Yaskawa INFORM job: OK_R2_O55A(90,180)KMOK_HARDOX.JBI

/JOB
//NAME OK_R2_O55A(90,180)KMOK_HARDOX
//POS
///NPOS 281,281,281,21,0,0
///TOOL 0
///POSTYPE PULSE
///PULSE
C00000=-111506,-49155,-65609,8484,85356,-77443
C00001=-115517,55698,23689,9444,84726,-78820
C00002=-108924,22008,-28178,-1197,90006,-78517
C00003=-108800,12121,-29647,4496,81806,-65930
C00004=-108630,12702,-28416,4432,81339,-65891
C00005=-108630,12328,-27828,4436,80786,-65911
C00006=-108630,12408,-27956,4436,80905,-65905
C00007=-108261,14534,-26027,4289,80792,-65794
C00008=-108630,12408,-27956,4436,80905,-65905
C00009=-107811,11629,-28656,4106,80897,-65648
C00010=-106858,10805,-29394,3723,80886,-65349
C00011=-107811,12739,-30286,4093,82467,-65597
C00012=-109010,42723,-6645,1454,97503,-73185
C00013=-109059,41996,-5623,1462,96501,-73210
C00014=-109059,41520,-5019,1461,95884,-73214
C00015=-109059,41606,-5129,1461,95997,-73214
C00016=-109349,39393,-7454,1528,96295,-73302
C00017=-109059,41606,-5129,1461,95997,-73214
C00018=-105960,29621,-15205,-5152,89122,-73169
C00019=-106826,30438,-14390,-4880,88993,-73434
C00020=-106699,31092,-15669,-4922,90120,-73439
C00021=-111304,-6970,-55605,-8918,107850,-76513
C00022=-101629,-20179,-65627,-10374,108234,-73505
C00023=-102461,-22935,-63329,-10075,105355,-73520
C00024=-102461,-23546,-62650,-10036,104633,-73460
C00025=-102461,-23453,-62757,-10042,104746,-73469
C00026=-102879,-26170,-64656,-9970,104475,-73577
C00027=-102461,-23453,-62757,-10042,104746,-73469
C00028=-99476,-55184,-78355,-14129,83990,-71244
C00029=-100829,-54344,-77892,-13696,83914,-71680
C00030=-99476,-54678,-79370,-14114,84849,-71342
C00031=-104557,-74568,-89383,-2164,74355,-70375
C00032=-103806,-74176,-87211,-2482,73240,-70100
C00033=-103806,-74372,-86383,-2489,72630,-70088
C00034=-103806,-74333,-86558,-2489,72756,-70088
C00035=-103548,-71014,-84973,-2584,73493,-70016
C00036=-103806,-74333,-86558,-2489,72756,-70088
C00037=-102597,-74952,-86848,-2986,72658,-69674
C00038=-101312,-75790,-87238,-3514,72521,-69232
C00039=-102597,-74499,-88609,-2967,73972,-69706
C00040=-118555,-42842,-73429,3462,80943,-74869
C00041=-119429,-43574,-71478,3824,79408,-75190
C00042=-119429,-43990,-70690,3831,78712,-75212
C00043=-119429,-43899,-70866,3830,78866,-75207
C00044=-122277,-43888,-70860,4961,79012,-76114
C00045=-122277,-44025,-70591,4964,78778,-76124
C00046=-121086,-44057,-70608,4493,78709,-75744
C00047=-121531,-43284,-72024,4653,79998,-75839
C00048=-117272,-117266,-105575,3266,62469,-74939
C00049=-116519,-127007,-107880,3037,58859,-74752
C00050=-116519,-126380,-106487,3053,58326,-74766
C00051=-116519,-126568,-106901,3048,58484,-74761
C00052=-121865,-126759,-106958,5473,58705,-76855
C00053=-121865,-126441,-106262,5489,58442,-76869
C00054=-119655,-126444,-106264,4491,58305,-76004
C00055=-119655,-127215,-107960,4461,58951,-75978
C00056=-112812,-150066,-114118,1491,50753,-73411
C00057=-112812,-148729,-112487,1496,50436,-73414
C00058=-113217,-142059,-110816,1647,52843,-73550
C00059=-113131,-144600,-112664,1608,52672,-73518
C00060=-64818,-116281,-103066,-23997,61655,-54736
C00061=-62465,-114100,-100180,-25084,61755,-53781
C00062=-62465,-113608,-98707,-25230,61158,-53639
C00063=-62465,-113710,-99005,-25201,61277,-53666
C00064=-58836,-120022,-101046,-27063,60627,-51963
C00065=-58836,-119826,-100588,-27108,60466,-51920
C00066=-60233,-117500,-99850,-26399,60681,-52575
C00067=-60033,-118628,-101973,-26303,61399,-52670
C00068=-95049,-20989,-71107,5943,107094,-67526
C00069=-77423,-912,-56771,2322,107833,-62256
C00070=-76072,-2112,-53613,2004,105243,-61899
C00071=-76072,-2916,-53031,1997,104470,-61910
C00072=-76072,-2789,-53124,1997,104594,-61910
C00073=-75971,-5189,-55074,1975,104559,-61882
C00074=-76072,-2789,-53124,1997,104594,-61910
C00075=-72991,-17697,-62638,-2229,94769,-69319
C00076=-74281,-17927,-62808,-1837,94727,-69700
C00077=-72991,-16562,-63565,-2235,95923,-69339
C00078=-75226,-46418,-75690,9290,73375,-84742
C00079=-74182,-46690,-75145,8802,72795,-84444
C00080=-74182,-47182,-74296,8836,72029,-84500
C00081=-74182,-47096,-74453,8830,72169,-84490
C00082=-74244,-44038,-72629,8839,72620,-84478
C00083=-74182,-47096,-74453,8830,72169,-84490
C00084=-73094,-46764,-74257,8291,72112,-84135
C00085=-72074,-46719,-74230,7784,72025,-83806
C00086=-72401,-46093,-76320,7882,73648,-83808
C00087=-67489,-6166,-61905,14115,111060,-76264
C00088=-69649,20522,-33673,24556,114676,-73904
C00089=-69671,18738,-32349,24199,113097,-74275
C00090=-69671,18146,-31824,24077,112524,-74402
C00091=-69671,18262,-31932,24102,112638,-74377
C00092=-69800,17846,-32320,24118,112695,-74410
C00093=-69675,18599,-32561,24211,113152,-74264
C00094=-63225,2541,-47955,23753,112661,-72111
C00095=-63277,1683,-47440,23617,111977,-72278
C00096=-63277,1073,-46916,23502,111394,-72405
C00097=-63277,1203,-47030,23526,111518,-72377
C00098=-63425,725,-47430,23545,111556,-72420
C00099=-63342,1826,-48065,23712,112415,-72205
C00100=-62206,17260,-37784,17009,103305,-74838
C00101=-61339,16149,-35110,16634,101032,-74890
C00102=-61339,15490,-34544,16589,100372,-74981
C00103=-61339,15587,-34628,16595,100471,-74968
C00104=-60359,16269,-33999,16356,100262,-74691
C00105=-61339,15587,-34628,16595,100471,-74968
C00106=-61066,13263,-36755,16538,100533,-74873
C00107=-60785,11321,-38512,16476,100561,-74782
C00108=-61066,13913,-37304,16583,101180,-74784
C00109=-55537,11439,-40793,10264,96708,-89931
C00110=-55386,12069,-40617,10225,96903,-89870
C00111=-55386,11332,-40052,10205,96188,-89929
C00112=-55386,11448,-40144,10209,96302,-89918
C00113=-56455,10727,-40790,10532,96446,-90224
C00114=-55386,11448,-40144,10209,96302,-89918
C00115=-55615,12989,-38751,10276,96262,-89989
C00116=-56013,15101,-36821,10392,96204,-90111
C00117=-55930,15302,-38056,10390,97045,-90015
C00118=-69610,-27139,-66329,21663,80743,-86076
C00119=-68739,-29162,-64945,21405,78779,-86142
C00120=-68739,-29645,-64290,21446,78173,-86252
C00121=-68739,-29425,-64595,21426,78455,-86201
C00122=-70305,-29836,-64873,22111,78793,-86664
C00123=-70305,-30098,-64507,22135,78458,-86726
C00124=-69784,-29812,-64314,21908,78356,-86568
C00125=-70093,-29888,-65249,22006,78930,-86565
C00126=-69460,-16189,-57169,21614,80708,-86031
C00127=-69490,-16804,-56284,21674,79908,-86184
C00128=-69490,-17306,-55650,21712,79303,-86294
C00129=-69490,-16804,-56284,21674,79908,-86184
C00130=-71198,-17146,-56538,22415,80299,-86675
C00131=-71198,-17694,-55840,22455,79641,-86800
C00132=-70522,-17552,-55735,22163,79484,-86605
C00133=-70652,-17250,-56551,22180,80125,-86528
C00134=-59067,-8187,-54664,-1101,82113,-86494
C00135=-58982,-12091,-55682,-1142,80734,-86460
C00136=-58982,-12659,-55089,-1143,80077,-86456
C00137=-58982,-12365,-55400,-1142,80420,-86459
C00138=-58542,-15777,-57986,-1343,80263,-86324
C00139=-58542,-16216,-57517,-1344,79752,-86321
C00140=-58731,-14747,-56416,-1258,79827,-86379
C00141=-58929,-14817,-58024,-1165,80777,-86449
C00142=-74865,-14118,-62828,-14130,92718,-81050
C00143=-74988,-16459,-62145,-14059,91123,-80906
C00144=-74988,-17205,-61497,-14051,90361,-80819
C00145=-74988,-16814,-61843,-14056,90763,-80864
C00146=-74878,-20571,-64590,-14091,90545,-80806
C00147=-74878,-21004,-64202,-14087,90099,-80754
C00148=-75042,-19403,-63044,-14030,90184,-80814
C00149=-74977,-18175,-64416,-14070,91627,-80958
C00150=-70693,-7790,-53035,631,77874,-74575
C00151=-70154,-9444,-51202,364,75895,-74417
C00152=-70154,-9889,-50670,365,75339,-74418
C00153=-70154,-9794,-50790,365,75461,-74418
C00154=-70309,-7210,-48753,442,75536,-74465
C00155=-70154,-9794,-50790,365,75461,-74418
C00156=-69601,-9613,-50649,89,75466,-74246
C00157=-68418,-9035,-50194,-503,75489,-73877
C00158=-70154,-8777,-51949,363,76695,-74414
C00159=-72134,44695,-6984,-4762,104287,-75834
C00160=-72134,44301,-6603,-4750,103850,-75816
C00161=-72134,43688,-5973,-4734,103152,-75788
C00162=-72134,43787,-6082,-4735,103269,-75794
C00163=-72123,41447,-8571,-4742,103595,-75805
C00164=-72134,43787,-6082,-4735,103270,-75794
C00165=-73005,43598,-6282,-4599,103251,-76067
C00166=-73786,43384,-6510,-4475,103242,-76313
C00167=-73018,44528,-7213,-4622,104298,-76111
C00168=-79422,35817,-13411,7006,100751,-75778
C00169=-74570,36341,-12845,6044,100322,-74293
C00170=-74570,36341,-12845,6044,100322,-74293
C00171=-72929,24013,-22984,4225,91927,-74293
C00172=-70584,14325,-29595,-1089,84518,-74676
C00173=-68494,21486,-24488,-6892,89276,-75326
C00174=-69395,21903,-23934,-10573,89960,-76456
C00175=-69395,21903,-23934,-10573,89960,-76456
C00176=-71080,32446,-16078,-8958,97674,-77386
C00177=-79422,35817,-13411,7006,100751,-75778
C00178=-79438,36883,-13685,7031,101465,-75742
C00179=-62206,17260,-37784,17009,103305,-74838
C00180=-61339,16149,-35110,16634,101032,-74890
C00181=-60712,-19322,-56729,15368,77567,-77605
C00182=-59094,-21751,-57339,14674,76450,-77219
C00183=-61038,-23011,-55706,17436,71746,-78177
C00184=-62083,-14156,-49199,17905,72476,-78422
C00185=-62083,-14156,-49199,17905,72476,-78422
C00186=-57090,11564,-36742,7182,90651,-76876
C00187=-56002,36932,-16764,6614,106870,-88572
C00188=-52140,41844,-13688,6040,107237,-87347
C00189=-48975,42648,-12828,5535,106926,-86378
C00190=-48975,42648,-12828,5535,106926,-86378
C00191=-52691,32805,-21114,13853,102301,-85620
C00192=-59094,-21751,-57339,14674,76450,-77219
C00193=-59425,-21539,-59164,14761,77698,-77175
C00194=-82076,-56968,-83798,24635,79831,-84346
C00195=-77747,-24152,-67705,18938,100689,-79924
C00196=-78057,-28160,-69137,18928,99634,-80190
C00197=-70869,-26802,-68287,17174,98411,-78082
C00198=-70869,-26802,-68287,17174,98411,-78082
C00199=-62364,-43762,-77635,6437,85665,-78480
C00200=-58442,-42143,-76885,-289,85725,-78490
C00201=-56915,-39089,-75695,-4701,88717,-80179
C00202=-58604,-34961,-73950,-7014,92707,-81523
C00203=-58604,-34961,-73950,-7014,92707,-81523
C00204=-58166,-35258,-74455,-8537,94295,-81804
C00205=-78057,-28160,-69137,18928,99634,-80190
C00206=-78109,-26468,-70352,19060,101178,-79960
C00207=-101629,-20179,-65627,-10374,108234,-73505
C00208=-103344,-22647,-63272,-9953,105369,-73804
C00209=-103510,-25764,-64254,-9875,104364,-73776
C00210=-96684,-29558,-66841,-10807,104795,-71624
C00211=-96684,-29558,-66841,-10807,104795,-71624
C00212=-95283,-51624,-78295,-10520,89912,-69715
C00213=-89288,-71016,-83236,-19331,74161,-66844
C00214=-92735,-73848,-83866,-17944,70715,-67525
C00215=-98754,-71520,-82752,-15362,70010,-69594
C00216=-98754,-71520,-82752,-15362,70010,-69594
C00217=-103983,-45462,-74593,-9714,90020,-72843
C00218=-103510,-25764,-64254,-9875,104364,-73776
C00219=-103560,-24307,-64999,-9933,105549,-73890
C00220=-69649,20522,-33673,24556,114676,-73904
C00221=-71557,26749,-25386,24354,113424,-74867
C00222=-68289,18895,-32791,17896,110504,-75619
C00223=-68202,19061,-32635,17883,110476,-75594
C00224=-68581,18341,-33310,17936,110593,-75702
C00225=-67453,16954,-34605,17788,110459,-75347
C00226=-67453,17755,-35235,17895,111222,-75226
C00227=-59289,756,-51060,6867,103388,-84120
C00228=-56748,-5812,-54346,2389,98605,-84475
C00229=-64645,12200,-39595,15963,109468,-83302
C00230=-61225,2939,-46046,22972,113017,-79913
C00231=-60681,1709,-47088,22917,112895,-79749
C00232=-58469,-3087,-51074,22687,112356,-79091
C00233=-58469,-1901,-52028,22910,113464,-78859
C00234=-117837,-87974,-96376,3289,71861,-74881
C00235=-92533,-132854,-111618,-21009,63789,-66049
C00236=-78523,-139004,-102182,-39306,54450,-56561
C00237=-81657,-141710,-102852,-38814,52284,-57229
C00238=-81657,-141710,-102852,-38814,52284,-57229
C00239=-114174,-154940,-107271,-2509,34053,-71746
C00240=-140780,-145696,-102896,33687,43289,-86686
C00241=-138023,-130656,-99106,29500,46903,-83798
C00242=-128713,-21741,-47637,18171,66698,-75148
C00243=-128713,-20196,-51555,17794,69753,-74669
C00244=-109059,43195,-6970,1468,97945,-73193
C00245=-113001,46227,-1101,7447,98334,-73296
C00246=-113396,48521,2242,7746,99771,-73296
C00247=-109170,43506,-3227,7034,100204,-71930
C00248=-109170,43506,-3227,7034,100204,-71930
C00249=-110675,25111,-18338,12830,89041,-80433
C00250=-106850,7079,-30449,5687,75314,-81784
C00251=-105360,10734,-28025,177,76815,-82287
C00252=-108676,13612,-25432,1655,76734,-83345
C00253=-108676,13612,-25432,1655,76734,-83345
C00254=-107152,30192,-14315,-2638,88634,-83622
C00255=-113396,48521,2242,7746,99771,-73296
C00256=-113396,49658,801,7791,101229,-73204
C00257=-101766,-98767,-99644,-3411,68336,-69273
C00258=-70067,-34207,-71053,21900,80175,-86329
C00259=-68941,-37910,-69134,21595,77036,-86529
C00260=-69099,-37316,-68757,21658,77143,-86564
C00261=-69654,-30548,-64331,21843,77979,-86598
C00262=-70579,-15119,-53564,22144,79419,-86640
C00263=-70579,-15119,-53564,22144,79419,-86640
C00264=-59362,-1592,-48978,2748,88384,-85470
C00265=-54202,-4221,-50196,-5979,86559,-88824
C00266=-54998,-5045,-50841,-6864,86759,-89370
C00267=-54493,-339,-47792,-12989,90949,-86203
C00268=-70768,-8822,-54873,-7152,89179,-90922
C00269=-60817,-19294,-55988,-26592,80523,-79978
C00270=-60817,-16249,-59555,-26407,83905,-80744
C00271=-62218,-50547,-80619,-18317,72013,-76735
C00272=-117272,-117266,-105575,3266,62469,-74939
C00273=-127230,-85492,-91646,16880,70768,-77338
C00274=-127349,-94743,-89409,19343,58411,-79334
C00275=-124353,-95100,-89551,17820,57640,-78233
C00276=-84234,-78954,-82744,-5379,58597,-62424
C00277=-80328,-74945,-80894,-7540,59821,-60991
C00278=-80936,-76895,-83460,-7157,60340,-61258
C00279=-73139,-123053,-107935,-12603,52748,-57405
C00280=-44833,-55261,-28957,-41445,79036,76616
BC00000=282524,663602,181971
BC00001=288445,778354,181971
BC00002=288445,813516,60117
BC00003=288445,813516,60117
BC00004=288445,813515,60114
BC00005=288445,813515,60114
BC00006=288445,813515,60114
BC00007=288445,813515,60114
BC00008=288445,813515,60114
BC00009=288445,813515,60114
BC00010=288445,813515,60114
BC00011=288445,813515,60114
BC00012=288445,813515,60114
BC00013=288445,813515,60114
BC00014=288445,813515,60114
BC00015=288445,813515,60114
BC00016=288445,813515,60114
BC00017=288445,813515,60114
BC00018=288445,813515,60114
BC00019=288445,813515,60114
BC00020=288445,813515,60114
BC00021=288445,813515,60114
BC00022=288445,813515,60114
BC00023=288445,813515,60114
BC00024=288445,813515,60114
BC00025=288445,813515,60114
BC00026=288445,813515,60114
BC00027=288445,813515,60114
BC00028=288445,813515,60114
BC00029=288445,813515,60114
BC00030=288445,813515,60114
BC00031=288445,813515,60114
BC00032=288445,813515,60114
BC00033=288445,813515,60114
BC00034=288445,813515,60114
BC00035=288445,813515,60114
BC00036=288445,813515,60114
BC00037=288445,813515,60114
BC00038=288445,813515,60114
BC00039=288445,813515,60114
BC00040=288445,813515,60113
BC00041=288445,813515,60113
BC00042=288445,813515,60113
BC00043=288445,813515,60113
BC00044=288445,813515,60113
BC00045=288445,813515,60113
BC00046=288445,813515,60113
BC00047=288445,813515,60113
BC00048=286846,785286,60113
BC00049=286846,785286,60113
BC00050=286846,785286,60113
BC00051=286846,785286,60113
BC00052=286846,785286,60113
BC00053=286846,785286,60113
BC00054=286846,785286,60113
BC00055=286846,785286,60113
BC00056=286846,785286,60113
BC00057=286846,785286,60113
BC00058=286846,785286,60113
BC00059=286846,785286,60113
BC00060=286846,785286,60113
BC00061=286846,785286,60113
BC00062=286846,785286,60113
BC00063=286846,785286,60113
BC00064=286846,785286,60113
BC00065=286846,785286,60113
BC00066=286846,785286,60113
BC00067=286846,785286,60113
BC00068=286846,785286,60113
BC00069=256051,786407,19658
BC00070=256051,786407,19658
BC00071=256051,786407,19658
BC00072=256051,786407,19658
BC00073=256051,786407,19658
BC00074=256051,786407,19658
BC00075=256051,786407,19658
BC00076=256051,786407,19658
BC00077=256051,786407,19658
BC00078=256051,786407,19658
BC00079=256051,786407,19658
BC00080=256051,786407,19658
BC00081=256051,786407,19658
BC00082=256051,786407,19658
BC00083=256051,786407,19658
BC00084=256051,786407,19658
BC00085=256051,786407,19658
BC00086=256051,786407,19658
BC00087=249253,815901,19362
BC00088=249253,815901,19362
BC00089=249253,815901,19362
BC00090=249253,815901,19362
BC00091=249253,815901,19362
BC00092=249253,815901,19362
BC00093=249253,815901,19362
BC00094=249253,815901,19362
BC00095=249253,815901,19362
BC00096=249253,815901,19362
BC00097=249253,815901,19362
BC00098=249253,815901,19362
BC00099=249253,815901,19362
BC00100=249253,815901,19362
BC00101=249253,815901,19362
BC00102=249253,815901,19362
BC00103=249253,815901,19362
BC00104=249253,815901,19362
BC00105=249253,815901,19362
BC00106=249253,815901,19362
BC00107=249253,815901,19362
BC00108=249253,815901,19362
BC00109=249253,822904,11778
BC00110=249253,822904,9053
BC00111=249253,822904,9053
BC00112=249253,822904,9053
BC00113=249253,822904,9053
BC00114=249253,822904,9053
BC00115=249253,822904,9053
BC00116=249253,822904,9053
BC00117=249253,822904,9053
BC00118=249254,822904,9050
BC00119=249254,822904,9050
BC00120=249254,822904,9050
BC00121=249254,822904,9050
BC00122=249254,822904,9050
BC00123=249254,822904,9050
BC00124=249254,822904,9050
BC00125=249254,822904,9050
BC00126=249254,822904,9050
BC00127=249254,822904,9050
BC00128=249254,822904,9050
BC00129=249254,822904,9050
BC00130=249254,822904,9050
BC00131=249254,822904,9050
BC00132=249254,822904,9050
BC00133=249254,822904,9050
BC00134=249254,822904,9050
BC00135=249254,822904,9050
BC00136=249254,822904,9050
BC00137=249254,822904,9050
BC00138=249254,822904,9050
BC00139=249254,822904,9050
BC00140=249254,822904,9050
BC00141=249254,822904,9050
BC00142=278045,822904,9050
BC00143=278045,822904,9050
BC00144=278045,822904,9050
BC00145=278045,822904,9050
BC00146=278045,822904,9050
BC00147=278045,822904,9050
BC00148=278045,822904,9050
BC00149=278045,822904,9050
BC00150=278045,822904,9047
BC00151=278045,822904,9047
BC00152=278045,822904,9047
BC00153=278045,822904,9047
BC00154=278045,822904,9047
BC00155=278045,822904,9047
BC00156=278045,822904,9047
BC00157=278045,822904,9047
BC00158=278045,822904,9047
BC00159=278045,813873,46918
BC00160=278045,813873,46918
BC00161=278045,813873,46918
BC00162=278045,813873,46918
BC00163=278045,813873,46918
BC00164=278045,813873,46918
BC00165=278045,813873,46918
BC00166=278045,813873,46918
BC00167=278045,813873,46918
BC00168=278045,813873,46918
BC00169=278045,813873,46918
BC00170=278045,813873,46918
BC00171=278045,813873,46918
BC00172=278045,813873,46918
BC00173=278045,813873,46918
BC00174=278045,813873,46918
BC00175=278045,813873,46918
BC00176=278045,813873,46918
BC00177=278045,813873,46918
BC00178=278045,813873,46918
BC00179=249253,815901,19362
BC00180=249253,815901,19362
BC00181=249254,815900,19361
BC00182=249254,815900,19361
BC00183=249325,815895,19429
BC00184=249325,815895,19429
BC00185=249325,815895,19429
BC00186=249325,815895,19429
BC00187=249325,815895,19429
BC00188=235058,815895,6680
BC00189=224411,815895,6680
BC00190=224411,815895,6680
BC00191=224412,815895,6676
BC00192=249254,815900,19361
BC00193=249254,815900,19361
BC00194=249254,815900,19361
BC00195=249254,815900,19360
BC00196=249254,815900,19360
BC00197=249306,815896,19410
BC00198=249306,815896,19410
BC00199=249306,815896,19410
BC00200=249306,815896,19410
BC00201=249339,815894,19441
BC00202=249339,815894,19441
BC00203=249339,815894,19441
BC00204=249339,815894,19441
BC00205=249254,815900,19360
BC00206=249254,815900,19360
BC00207=288445,813515,60114
BC00208=288445,813515,60114
BC00209=288445,813515,60114
BC00210=288439,813515,60106
BC00211=288439,813515,60106
BC00212=288439,813515,60106
BC00213=288439,813515,60106
BC00214=288432,813515,60098
BC00215=288432,813515,60098
BC00216=288432,813515,60098
BC00217=288432,813515,60098
BC00218=288445,813515,60114
BC00219=288445,813515,60114
BC00220=249253,815901,19362
BC00221=249254,815901,19362
BC00222=249254,815901,19362
BC00223=249254,815901,19362
BC00224=249254,815901,19362
BC00225=249254,815900,19361
BC00226=249254,815900,19361
BC00227=249254,815900,19361
BC00228=249254,815900,19361
BC00229=249254,815900,19361
BC00230=249254,815900,19361
BC00231=249254,815900,19361
BC00232=249254,815900,19361
BC00233=249254,815900,19361
BC00234=288445,813515,60113
BC00235=288445,781013,60113
BC00236=288445,781013,60113
BC00237=288445,781013,60113
BC00238=288445,781013,60113
BC00239=288445,781013,60113
BC00240=288445,781013,60113
BC00241=288445,781013,60113
BC00242=288445,781013,60113
BC00243=288445,781013,60113
BC00244=288445,813515,60114
BC00245=288445,813515,60114
BC00246=288445,813515,60114
BC00247=288445,813515,60114
BC00248=288445,813515,60114
BC00249=288445,813515,60114
BC00250=288445,813515,60114
BC00251=288445,813515,60114
BC00252=288445,813515,60114
BC00253=288445,813515,60114
BC00254=288445,813515,60114
BC00255=288445,813515,60114
BC00256=288445,813515,60114
BC00257=288445,813515,60114
BC00258=249254,822904,9050
BC00259=249255,822904,9046
BC00260=249255,822904,9046
BC00261=249255,822904,9046
BC00262=249255,822904,9045
BC00263=249255,822904,9045
BC00264=249255,822904,9045
BC00265=249255,822904,9045
BC00266=249255,822904,9045
BC00267=249255,822904,9045
BC00268=249255,822904,9045
BC00269=249255,822904,9045
BC00270=249255,822904,9045
BC00271=249255,822904,9045
BC00272=286846,785286,60113
BC00273=286846,744660,60113
BC00274=286846,744660,60113
BC00275=286846,744660,60113
BC00276=286797,744763,60046
BC00277=286797,744763,60046
BC00278=286797,744763,60046
BC00279=286797,744763,60046
BC00280=354635,666962,735004
EC00000=798156,1112951
EC00001=798156,1112951
EC00002=798156,1112951
EC00003=798156,1112951
EC00004=798155,1112951
EC00005=798155,1112951
EC00006=798155,1112951
EC00007=798155,1112951
EC00008=798155,1112951
EC00009=798155,1112951
EC00010=798155,1112951
EC00011=798155,1112951
EC00012=798155,1112951
EC00013=798155,1112951
EC00014=798155,1112951
EC00015=798155,1112951
EC00016=798155,1112951
EC00017=798155,1112951
EC00018=798155,1112951
EC00019=798155,1112951
EC00020=798155,1112951
EC00021=798155,1112951
EC00022=798155,1112951
EC00023=798155,1112951
EC00024=798155,1112951
EC00025=798155,1112951
EC00026=798155,1112951
EC00027=798155,1112951
EC00028=798155,1112951
EC00029=798155,1112951
EC00030=798155,1112951
EC00031=798155,1112951
EC00032=798155,1112951
EC00033=798155,1112951
EC00034=798155,1112951
EC00035=798155,1112951
EC00036=798155,1112951
EC00037=798155,1112951
EC00038=798155,1112951
EC00039=798155,1112951
EC00040=798153,1112950
EC00041=798153,1112950
EC00042=798153,1112950
EC00043=798153,1112950
EC00044=798153,1112950
EC00045=798153,1112950
EC00046=798153,1112950
EC00047=798153,1112950
EC00048=798153,1112950
EC00049=798153,1112950
EC00050=798153,1112950
EC00051=798153,1112950
EC00052=798153,1112950
EC00053=798153,1112950
EC00054=798153,1112950
EC00055=798153,1112950
EC00056=798153,1112950
EC00057=798153,1112950
EC00058=798153,1112950
EC00059=798153,1112950
EC00060=798153,1112950
EC00061=798153,1112950
EC00062=798153,1112950
EC00063=798153,1112950
EC00064=798153,1112950
EC00065=798153,1112950
EC00066=798153,1112950
EC00067=798153,1112950
EC00068=798153,1112950
EC00069=798153,1112950
EC00070=798153,1112950
EC00071=798153,1112950
EC00072=798153,1112950
EC00073=798153,1112950
EC00074=798153,1112950
EC00075=798153,1112950
EC00076=798153,1112950
EC00077=798153,1112950
EC00078=798153,1112950
EC00079=798153,1112950
EC00080=798153,1112950
EC00081=798153,1112950
EC00082=798153,1112950
EC00083=798153,1112950
EC00084=798153,1112950
EC00085=798153,1112950
EC00086=798153,1112950
EC00087=798152,1112949
EC00088=798152,1112949
EC00089=798152,1112949
EC00090=798152,1112949
EC00091=798152,1112949
EC00092=798152,1112949
EC00093=798152,1112949
EC00094=798152,1112949
EC00095=798152,1112949
EC00096=798152,1112949
EC00097=798152,1112949
EC00098=798152,1112949
EC00099=798152,1112949
EC00100=798152,1112949
EC00101=798152,1112949
EC00102=798152,1112949
EC00103=798152,1112949
EC00104=798152,1112949
EC00105=798152,1112949
EC00106=798152,1112949
EC00107=798152,1112949
EC00108=798152,1112949
EC00109=798152,1112949
EC00110=798152,1112949
EC00111=798152,1112949
EC00112=798152,1112949
EC00113=798152,1112949
EC00114=798152,1112949
EC00115=798152,1112949
EC00116=798152,1112949
EC00117=798152,1112949
EC00118=798151,1112948
EC00119=798150,1112947
EC00120=798150,1112947
EC00121=798150,1112947
EC00122=798150,1112947
EC00123=798150,1112947
EC00124=798150,1112947
EC00125=798150,1112947
EC00126=798150,1112947
EC00127=798150,1112947
EC00128=798150,1112947
EC00129=798150,1112947
EC00130=798150,1112947
EC00131=798150,1112947
EC00132=798150,1112947
EC00133=798150,1112947
EC00134=798150,1112947
EC00135=798150,1112947
EC00136=798150,1112947
EC00137=798150,1112947
EC00138=798150,1112947
EC00139=798150,1112947
EC00140=798150,1112947
EC00141=798150,1112947
EC00142=798150,1112947
EC00143=798150,1112947
EC00144=798150,1112947
EC00145=798150,1112947
EC00146=798150,1112947
EC00147=798150,1112947
EC00148=798150,1112947
EC00149=798150,1112947
EC00150=798148,1112946
EC00151=798148,1112946
EC00152=798148,1112946
EC00153=798148,1112946
EC00154=798148,1112946
EC00155=798148,1112946
EC00156=798148,1112946
EC00157=798148,1112946
EC00158=798148,1112946
EC00159=798148,1112946
EC00160=798148,1112946
EC00161=798148,1112946
EC00162=798148,1112946
EC00163=798148,1112946
EC00164=798148,1112946
EC00165=798148,1112946
EC00166=798148,1112946
EC00167=798148,1112946
EC00168=798148,1112946
EC00169=798148,1112946
EC00170=798148,1112946
EC00171=798148,1112946
EC00172=798148,1112946
EC00173=798148,1112946
EC00174=798148,1112946
EC00175=798148,1112946
EC00176=798148,1112946
EC00177=798148,1112946
EC00178=798148,1112946
EC00179=798152,1112949
EC00180=798152,1112949
EC00181=798151,1112948
EC00182=798151,1112948
EC00183=798151,1112948
EC00184=798151,1112948
EC00185=798151,1112948
EC00186=798151,1112948
EC00187=798151,1112948
EC00188=798151,1112948
EC00189=798151,1112948
EC00190=798151,1112948
EC00191=798150,1112947
EC00192=798151,1112948
EC00193=798151,1112948
EC00194=798151,1112948
EC00195=798150,1112947
EC00196=798150,1112947
EC00197=798150,1112947
EC00198=798150,1112947
EC00199=798150,1112947
EC00200=798150,1112947
EC00201=798150,1112947
EC00202=798150,1112947
EC00203=798150,1112947
EC00204=798150,1112947
EC00205=798150,1112947
EC00206=798150,1112947
EC00207=798155,1112951
EC00208=798155,1112951
EC00209=798155,1112951
EC00210=798155,1112951
EC00211=798155,1112951
EC00212=798155,1112951
EC00213=798155,1112951
EC00214=798155,1112951
EC00215=798155,1112951
EC00216=798155,1112951
EC00217=798155,1112951
EC00218=798155,1112951
EC00219=798155,1112951
EC00220=798152,1112949
EC00221=798151,1112948
EC00222=798151,1112948
EC00223=798151,1112948
EC00224=798151,1112948
EC00225=798150,1112948
EC00226=798150,1112948
EC00227=798150,1112948
EC00228=798150,1112948
EC00229=798150,1112948
EC00230=798150,1112948
EC00231=798150,1112948
EC00232=798150,1112948
EC00233=798150,1112948
EC00234=798153,1112950
EC00235=798153,1112950
EC00236=798153,1112950
EC00237=798153,1112950
EC00238=798153,1112950
EC00239=798153,1112950
EC00240=798153,1112950
EC00241=798153,1112950
EC00242=798153,1112950
EC00243=798153,1112950
EC00244=798155,1112951
EC00245=798155,1112951
EC00246=798155,1112951
EC00247=798155,1112951
EC00248=798155,1112951
EC00249=798155,1112951
EC00250=798155,1112951
EC00251=798155,1112951
EC00252=798155,1112951
EC00253=798155,1112951
EC00254=798155,1112951
EC00255=798155,1112951
EC00256=798155,1112951
EC00257=798155,1112951
EC00258=798151,1112948
EC00259=798150,1112947
EC00260=798150,1112947
EC00261=798150,1112947
EC00262=798149,1112946
EC00263=798149,1112946
EC00264=798149,1112946
EC00265=798149,1112946
EC00266=798149,1112946
EC00267=798149,1112946
EC00268=798149,1112946
EC00269=798149,1112946
EC00270=798149,1112946
EC00271=798149,1112946
EC00272=798153,1112950
EC00273=798153,1112950
EC00274=798153,1112950
EC00275=798153,1112950
EC00276=798153,1112950
EC00277=798153,1112950
EC00278=798153,1112950
EC00279=798153,1112950
EC00280=798156,1112951
///POSTYPE BASE
///RECTAN
///RCONF 0,0,0,0,0,0,0,0,0,0,0,0,0,0,0,0,0,0,0,0,0,0,0,0
P00006=0.222,-3.123,-1.508,0.0000,0.0000,0.0000
P00021=-0.225,-6.128,-0.405,0.0000,0.0000,0.0000
P00022=0.222,-3.123,-1.508,0.0000,0.0000,0.0000
P00023=0.143,-0.036,0.682,0.0000,0.0000,0.0000
P00024=0.145,-0.552,1.326,0.0000,0.0000,0.0000
P00025=-2.003,0.006,0.728,0.0000,0.0000,0.0000
P00026=0.562,-0.002,-0.337,0.0000,0.0000,0.0000
P00027=-0.746,0.015,-9.096,0.0000,0.0000,0.0000
P00028=-2.237,-0.018,-7.702,0.0000,0.0000,0.0000
P00029=-2.156,-0.086,-4.681,0.0000,0.0000,0.0000
P00030=5.926,-4.294,-1.390,0.0000,0.0000,0.0000
P00031=1.853,-0.001,-1.549,0.0000,0.0000,0.0000
P00032=1.957,0.503,-7.217,0.0000,0.0000,0.0000
///RCONF 0,0,0,0,1,0,0,0,0,0,0,0,0,0,0,0,0,0,0,0,0,0,0,0
P00033=-0.123,0.612,-5.012,0.0000,0.0000,0.0000
///RCONF 0,0,0,0,0,0,0,0,0,0,0,0,0,0,0,0,0,0,0,0,0,0,0,0
P00034=-0.304,0.773,-2.693,0.0000,0.0000,0.0000
P00035=2.817,0.591,-1.622,0.0000,0.0000,0.0000
P00036=-1.108,-0.829,1.850,0.0000,0.0000,0.0000
P00037=0.023,0.937,-2.677,0.0000,0.0000,0.0000
P00038=0.158,-1.133,-1.952,0.0000,0.0000,0.0000
P00039=0.012,-3.081,-0.106,0.0000,0.0000,0.0000
P00040=-0.030,9.648,2.467,0.0000,0.0000,0.0000
//INST
///DATE 2025/02/20 14:32
///ATTR SC,RW
///GROUP1 RB1,BS1
///GROUP2 ST1
NOP
'MUZYLO 300124
'MUZYLO 310124
'POPRAWA I SPAWANIE
'OK_R2_o55a(90,180)
'Path S3739
SFTOF3D
CALL JOB:CLEAN-R1_KM_3P
MOVJ C00000 BC00000 VJ=100.00  +MOVJ EC00000 VJ=100.00
MOVL C00001 BC00001 V=666.7  +MOVJ EC00001 VJ=100.00
MOVL C00002 BC00002 V=666.7  +MOVJ EC00002 VJ=100.00
MOVL C00003 BC00003 V=666.7  +MOVJ EC00003 VJ=100.00
SMOVL C00004 BC00004 V=166.7  +MOVJ EC00004
SREFP 3 C00005 BC00005  +REFP EC00005
CALL JOB:SEARCH-R1-S13D
SET P021 P006
SFTON3D P021
SMOVL C00006 BC00006 V=166.7  +MOVJ EC00006
SREFP 3 C00007 BC00007  +REFP EC00007
CALL JOB:SEARCH-R1-S13D
SET P021 P006
SFTON3D P021
SMOVL C00008 BC00008 V=166.7  +MOVJ EC00008
SMOVL C00009 BC00009 V=166.7  +MOVJ EC00009
SREFP 3 C00010 BC00010  +REFP EC00010
CALL JOB:SEARCH-R1-S13D
SET P021 P006
SFTON3D P021
SMOVL C00011 BC00011 V=166.7  +MOVJ EC00011
MOVL C00012 BC00012 V=666.7  +MOVJ EC00012 VJ=100.00
SMOVL C00013 BC00013 V=166.7  +MOVJ EC00013
SREFP 3 C00014 BC00014  +REFP EC00014
CALL JOB:SEARCH-R1-S13D
SET P022 P006
SFTON3D P022
SMOVL C00015 BC00015 V=166.7  +MOVJ EC00015
SREFP 3 C00016 BC00016  +REFP EC00016
CALL JOB:SEARCH-R1-S13D
SET P022 P006
SFTON3D P022
SMOVL C00017 BC00017 V=166.7  +MOVJ EC00017
SMOVL C00018 BC00018 V=166.7  +MOVJ EC00018
SREFP 3 C00019 BC00019  +REFP EC00019
CALL JOB:SEARCH-R1-S13D
SET P022 P006
SFTON3D P022
SMOVL C00020 BC00020 V=166.7  +MOVJ EC00020
SFTOF3D
MOVL C00021 BC00021 V=666.7  +MOVJ EC00021 VJ=100.00
MOVL C00022 BC00022 V=666.7  +MOVJ EC00022 VJ=100.00
SMOVL C00023 BC00023 V=166.7  +MOVJ EC00023
SREFP 3 C00024 BC00024  +REFP EC00024
CALL JOB:SEARCH-R1-S13D
SET P023 P006
SFTON3D P023
SMOVL C00025 BC00025 V=166.7  +MOVJ EC00025
SREFP 3 C00026 BC00026  +REFP EC00026
CALL JOB:SEARCH-R1-S13D
SET P023 P006
SFTON3D P023
SMOVL C00027 BC00027 V=166.7  +MOVJ EC00027
SMOVL C00028 BC00028 V=166.7  +MOVJ EC00028
SREFP 3 C00029 BC00029  +REFP EC00029
CALL JOB:SEARCH-R1-S13D
SET P023 P006
SFTON3D P023
SMOVL C00030 BC00030 V=166.7  +MOVJ EC00030
MOVL C00031 BC00031 V=666.7  +MOVJ EC00031 VJ=100.00
SMOVL C00032 BC00032 V=166.7  +MOVJ EC00032
SREFP 3 C00033 BC00033  +REFP EC00033
CALL JOB:SEARCH-R1-S13D
SET P024 P006
SFTON3D P024
SMOVL C00034 BC00034 V=166.7  +MOVJ EC00034
SREFP 3 C00035 BC00035  +REFP EC00035
CALL JOB:SEARCH-R1-S13D
SET P024 P006
SFTON3D P024
SMOVL C00036 BC00036 V=166.7  +MOVJ EC00036
SMOVL C00037 BC00037 V=166.7  +MOVJ EC00037
SREFP 3 C00038 BC00038  +REFP EC00038
CALL JOB:SEARCH-R1-S13D
SET P024 P006
SFTON3D P024
SMOVL C00039 BC00039 V=166.7  +MOVJ EC00039
SFTOF3D
MOVL C00040 BC00040 V=666.7  +MOVJ EC00040 VJ=100.00
SMOVL C00041 BC00041 V=166.7  +MOVJ EC00041
SREFP 3 C00042 BC00042  +REFP EC00042
CALL JOB:SEARCH-R1-S13D
SET P025 P006
SFTON3D P025
SMOVL C00043 BC00043 V=166.7  +MOVJ EC00043
SMOVL C00044 BC00044 V=166.7  +MOVJ EC00044
SMOVL C00045 BC00045 V=166.7  +MOVJ EC00045
SREFP 3 C00046 BC00046  +REFP EC00046
CALL JOB:SEARCH-R1-S13D
SET P025 P006
SFTON3D P025
SMOVL C00047 BC00047 V=166.7  +MOVJ EC00047
SFTOF3D
MOVL C00048 BC00048 V=666.7  +MOVJ EC00048 VJ=100.00
SMOVL C00049 BC00049 V=166.7  +MOVJ EC00049
SREFP 3 C00050 BC00050  +REFP EC00050
CALL JOB:SEARCH-R1-S13D
SET P026 P006
SFTON3D P026
SMOVL C00051 BC00051 V=166.7  +MOVJ EC00051
SMOVL C00052 BC00052 V=166.7  +MOVJ EC00052
SMOVL C00053 BC00053 V=166.7  +MOVJ EC00053
SREFP 3 C00054 BC00054  +REFP EC00054
CALL JOB:SEARCH-R1-S13D
SET P026 P006
SFTON3D P026
SMOVL C00055 BC00055 V=166.7  +MOVJ EC00055
SMOVL C00056 BC00056 V=166.7  +MOVJ EC00056
SMOVL C00057 BC00057 V=166.7  +MOVJ EC00057
SREFP 3 C00058 BC00058  +REFP EC00058
CALL JOB:SEARCH-R1-S13D
SET P027 P006
SFTON3D P027
SMOVL C00059 BC00059 V=166.7  +MOVJ EC00059
SFTOF3D
MOVL C00060 BC00060 V=666.7  +MOVJ EC00060 VJ=100.00
SMOVL C00061 BC00061 V=166.7  +MOVJ EC00061
SREFP 3 C00062 BC00062  +REFP EC00062
CALL JOB:SEARCH-R1-S13D
SET P028 P006
SFTON3D P028
SMOVL C00063 BC00063 V=166.7  +MOVJ EC00063
SMOVL C00064 BC00064 V=166.7  +MOVJ EC00064
SMOVL C00065 BC00065 V=166.7  +MOVJ EC00065
SREFP 3 C00066 BC00066  +REFP EC00066
CALL JOB:SEARCH-R1-S13D
SET P028 P006
SFTON3D P028
SMOVL C00067 BC00067 V=166.7  +MOVJ EC00067
SFTOF3D
SMOVL C00068 BC00068 V=666.7  +MOVJ EC00068
MOVL C00069 BC00069 V=666.7  +MOVJ EC00069 VJ=100.00
SMOVL C00070 BC00070 V=166.7  +MOVJ EC00070
SREFP 3 C00071 BC00071  +REFP EC00071
CALL JOB:SEARCH-R1-S13D
SET P029 P006
SFTON3D P029
SMOVL C00072 BC00072 V=166.7  +MOVJ EC00072
SREFP 3 C00073 BC00073  +REFP EC00073
CALL JOB:SEARCH-R1-S13D
SET P029 P006
SFTON3D P029
SMOVL C00074 BC00074 V=166.7  +MOVJ EC00074
SMOVL C00075 BC00075 V=166.7  +MOVJ EC00075
SREFP 3 C00076 BC00076  +REFP EC00076
CALL JOB:SEARCH-R1-S13D
SET P029 P006
SFTON3D P029
SMOVL C00077 BC00077 V=166.7  +MOVJ EC00077
MOVL C00078 BC00078 V=666.7  +MOVJ EC00078 VJ=100.00
SMOVL C00079 BC00079 V=166.7  +MOVJ EC00079
SREFP 3 C00080 BC00080  +REFP EC00080
CALL JOB:SEARCH-R1-S13D
SET P030 P006
SFTON3D P030
SMOVL C00081 BC00081 V=166.7  +MOVJ EC00081
SREFP 3 C00082 BC00082  +REFP EC00082
CALL JOB:SEARCH-R1-S13D
SET P030 P006
SFTON3D P030
SMOVL C00083 BC00083 V=166.7  +MOVJ EC00083
SMOVL C00084 BC00084 V=166.7  +MOVJ EC00084
SREFP 3 C00085 BC00085  +REFP EC00085
CALL JOB:SEARCH-R1-S13D
SET P030 P006
SFTON3D P030
SMOVL C00086 BC00086 V=166.7  +MOVJ EC00086
SMOVL C00087 BC00087 V=666.7  +MOVJ EC00087
SMOVL C00088 BC00088 V=666.7  +MOVJ EC00088
SMOVL C00089 BC00089 V=166.7  +MOVJ EC00089
SREFP 3 C00090 BC00090  +REFP EC00090
CALL JOB:SEARCH-R1-S13D
SET P031 P006
SFTON3D P031
SMOVL C00091 BC00091 V=166.7  +MOVJ EC00091
SREFP 3 C00092 BC00092  +REFP EC00092
CALL JOB:SEARCH-R1-S13D
SET P031 P006
SFTON3D P031
SMOVL C00093 BC00093 V=166.7  +MOVJ EC00093
SMOVL C00094 BC00094 V=666.7  +MOVJ EC00094
SMOVL C00095 BC00095 V=166.7  +MOVJ EC00095
SREFP 3 C00096 BC00096  +REFP EC00096
CALL JOB:SEARCH-R1-S13D
SET P032 P006
SFTON3D P032
SMOVL C00097 BC00097 V=166.7  +MOVJ EC00097
SREFP 3 C00098 BC00098  +REFP EC00098
CALL JOB:SEARCH-R1-S13D
SET P032 P006
SFTON3D P032
SMOVL C00099 BC00099 V=166.7  +MOVJ EC00099
SFTOF3D
MOVL C00100 BC00100 V=666.7  +MOVJ EC00100 VJ=100.00
SMOVL C00101 BC00101 V=166.7  +MOVJ EC00101
SREFP 3 C00102 BC00102  +REFP EC00102
CALL JOB:SEARCH-R1-S13D
SET P033 P006
SFTON3D P033
SMOVL C00103 BC00103 V=166.7  +MOVJ EC00103
SREFP 3 C00104 BC00104  +REFP EC00104
CALL JOB:SEARCH-R1-S13D
SET P033 P006
SFTON3D P033
SMOVL C00105 BC00105 V=166.7  +MOVJ EC00105
SMOVL C00106 BC00106 V=166.7  +MOVJ EC00106
SREFP 3 C00107 BC00107  +REFP EC00107
CALL JOB:SEARCH-R1-S13D
SET P033 P006
SFTON3D P033
SMOVL C00108 BC00108 V=166.7  +MOVJ EC00108
MOVL C00109 BC00109 V=666.7  +MOVJ EC00109 VJ=100.00
SMOVL C00110 BC00110 V=166.7  +MOVJ EC00110
SREFP 3 C00111 BC00111  +REFP EC00111
CALL JOB:SEARCH-R1-S13D
SET P034 P006
SFTON3D P034
SMOVL C00112 BC00112 V=166.7  +MOVJ EC00112
SREFP 3 C00113 BC00113  +REFP EC00113
CALL JOB:SEARCH-R1-S13D
SET P034 P006
SFTON3D P034
SMOVL C00114 BC00114 V=166.7  +MOVJ EC00114
SMOVL C00115 BC00115 V=166.7  +MOVJ EC00115
SREFP 3 C00116 BC00116  +REFP EC00116
CALL JOB:SEARCH-R1-S13D
SET P034 P006
SFTON3D P034
SMOVL C00117 BC00117 V=166.7  +MOVJ EC00117
MOVL C00118 BC00118 V=666.7  +MOVJ EC00118 VJ=0.78
SMOVL C00119 BC00119 V=166.7  +MOVJ EC00119
SREFP 3 C00120 BC00120  +REFP EC00120
CALL JOB:SEARCH-R1-S13D
SET P035 P006
SFTON3D P035
SMOVL C00121 BC00121 V=166.7  +MOVJ EC00121
SMOVL C00122 BC00122 V=166.7  +MOVJ EC00122
SMOVL C00123 BC00123 V=166.7  +MOVJ EC00123
SREFP 3 C00124 BC00124  +REFP EC00124
CALL JOB:SEARCH-R1-S13D
SET P035 P006
SFTON3D P035
SMOVL C00125 BC00125 V=166.7  +MOVJ EC00125
SMOVL C00126 BC00126 V=666.7  +MOVJ EC00126
SMOVL C00127 BC00127 V=166.7  +MOVJ EC00127
SREFP 3 C00128 BC00128  +REFP EC00128
CALL JOB:SEARCH-R1-S13D
SET P036 P006
SFTON3D P036
SMOVL C00129 BC00129 V=166.7  +MOVJ EC00129
SMOVL C00130 BC00130 V=166.7  +MOVJ EC00130
SMOVL C00131 BC00131 V=166.7  +MOVJ EC00131
SREFP 3 C00132 BC00132  +REFP EC00132
CALL JOB:SEARCH-R1-S13D
SET P036 P006
SFTON3D P036
SMOVL C00133 BC00133 V=166.7  +MOVJ EC00133
SMOVL C00134 BC00134 V=666.7  +MOVJ EC00134
SMOVL C00135 BC00135 V=166.7  +MOVJ EC00135
SREFP 3 C00136 BC00136  +REFP EC00136
CALL JOB:SEARCH-R1-S13D
SET P037 P006
SFTON3D P037
SMOVL C00137 BC00137 V=166.7  +MOVJ EC00137
SMOVL C00138 BC00138 V=166.7  +MOVJ EC00138
SMOVL C00139 BC00139 V=166.7  +MOVJ EC00139
SREFP 3 C00140 BC00140  +REFP EC00140
CALL JOB:SEARCH-R1-S13D
SET P037 P006
SFTON3D P037
SMOVL C00141 BC00141 V=166.7  +MOVJ EC00141
SMOVL C00142 BC00142 V=666.7  +MOVJ EC00142
SMOVL C00143 BC00143 V=166.7  +MOVJ EC00143
SREFP 3 C00144 BC00144  +REFP EC00144
CALL JOB:SEARCH-R1-S13D
SET P038 P006
SFTON3D P038
SMOVL C00145 BC00145 V=166.7  +MOVJ EC00145
SMOVL C00146 BC00146 V=166.7  +MOVJ EC00146
SMOVL C00147 BC00147 V=166.7  +MOVJ EC00147
SREFP 3 C00148 BC00148  +REFP EC00148
CALL JOB:SEARCH-R1-S13D
SET P038 P006
SFTON3D P038
SMOVL C00149 BC00149 V=166.7  +MOVJ EC00149
SMOVL C00150 BC00150 V=666.7  +MOVJ EC00150
SMOVL C00151 BC00151 V=166.7  +MOVJ EC00151
SREFP 3 C00152 BC00152  +REFP EC00152
CALL JOB:SEARCH-R1-S13D
SET P039 P006
SFTON3D P039
SMOVL C00153 BC00153 V=166.7  +MOVJ EC00153
SREFP 3 C00154 BC00154  +REFP EC00154
CALL JOB:SEARCH-R1-S13D
SET P039 P006
SFTON3D P039
SMOVL C00155 BC00155 V=166.7  +MOVJ EC00155
SMOVL C00156 BC00156 V=166.7  +MOVJ EC00156
SREFP 3 C00157 BC00157  +REFP EC00157
CALL JOB:SEARCH-R1-S13D
SET P039 P006
SFTON3D P039
SMOVL C00158 BC00158 V=166.7  +MOVJ EC00158
MOVL C00159 BC00159 V=666.7  +MOVJ EC00159 VJ=100.00
SMOVL C00160 BC00160 V=166.7  +MOVJ EC00160
SREFP 3 C00161 BC00161  +REFP EC00161
CALL JOB:SEARCH-R1-S13D
SET P040 P006
SFTON3D P040
SMOVL C00162 BC00162 V=166.7  +MOVJ EC00162
SREFP 3 C00163 BC00163  +REFP EC00163
CALL JOB:SEARCH-R1-S13D
SET P040 P006
SFTON3D P040
SMOVL C00164 BC00164 V=166.7  +MOVJ EC00164
SMOVL C00165 BC00165 V=166.7  +MOVJ EC00165
SREFP 3 C00166 BC00166  +REFP EC00166
CALL JOB:SEARCH-R1-S13D
SET P040 P006
SFTON3D P040
SMOVL C00167 BC00167 V=166.7  +MOVJ EC00167
MACRO1 MJ#(0) ARGF9
SMOVL C00168 BC00168 V=166.7 PL=0  +MOVJ EC00168
ARCON
SFTON3D P039
SMOVL C00169 BC00169 V=11.7  +MOVJ EC00169
SMOVC C00170 BC00170 V=15.0  +MOVJ EC00170
SMOVC C00171 BC00171 V=15.0  +MOVJ EC00171
SMOVC C00172 BC00172 V=15.0  +MOVJ EC00172
SFTON3D P040
SMOVL C00173 BC00173 V=11.7  +MOVJ EC00173
SMOVL C00174 BC00174 V=11.7  +MOVJ EC00174
SMOVC C00175 BC00175 V=15.0  +MOVJ EC00175
SMOVC C00176 BC00176 V=15.0  +MOVJ EC00176
SMOVC C00177 BC00177 V=15.0  +MOVJ EC00177
ARCOF
SMOVL C00178 BC00178 V=166.7  +MOVJ EC00178
SFTOF3D
MOVL C00179 BC00179 V=666.7  +MOVJ EC00179 VJ=100.00
SMOVL C00180 BC00180 V=166.7  +MOVJ EC00180
SMOVL C00181 BC00181 V=166.7  +MOVJ EC00181
SFTON3D P033
SMOVL C00182 BC00182 V=166.7 PL=0  +MOVJ EC00182
ARCON
SFTON3D P034
SMOVL C00183 BC00183 V=11.7  +MOVJ EC00183
SMOVL C00184 BC00184 V=11.7  +MOVJ EC00184
SMOVC C00185 BC00185 V=15.0  +MOVJ EC00185
SMOVC C00186 BC00186 V=15.0  +MOVJ EC00186
SMOVC C00187 BC00187 V=15.0  +MOVJ EC00187
SFTON3D P033
SMOVL C00188 BC00188 V=11.7  +MOVJ EC00188
SMOVL C00189 BC00189 V=11.7  +MOVJ EC00189
SMOVC C00190 BC00190 V=15.0  +MOVJ EC00190
SMOVC C00191 BC00191 V=15.0  +MOVJ EC00191
SMOVC C00192 BC00192 V=15.0  +MOVJ EC00192
ARCOF
SMOVL C00193 BC00193 V=166.7  +MOVJ EC00193
SFTOF3D
SMOVL C00194 BC00194 V=666.7  +MOVJ EC00194
SFTON3D P029
SMOVL C00195 BC00195 V=166.7  +MOVJ EC00195
SMOVL C00196 BC00196 V=166.7 PL=0  +MOVJ EC00196
ARCON
SFTON3D P030
SMOVL C00197 BC00197 V=11.7  +MOVJ EC00197
SMOVC C00198 BC00198 V=15.0  +MOVJ EC00198
SMOVC C00199 BC00199 V=15.0  +MOVJ EC00199
SMOVC C00200 BC00200 V=15.0  +MOVJ EC00200
SFTON3D P029
SMOVL C00201 BC00201 V=11.7  +MOVJ EC00201
SMOVL C00202 BC00202 V=11.7  +MOVJ EC00202
SMOVC C00203 BC00203 V=15.0  +MOVJ EC00203
SMOVC C00204 BC00204 V=15.0  +MOVJ EC00204
SMOVC C00205 BC00205 V=15.0  +MOVJ EC00205
ARCOF
SMOVL C00206 BC00206 V=166.7  +MOVJ EC00206
SFTOF3D
SMOVL C00207 BC00207 V=666.7  +MOVJ EC00207
SMOVL C00208 BC00208 V=666.7  +MOVJ EC00208
SFTON3D P023
SMOVL C00209 BC00209 V=166.7 PL=0  +MOVJ EC00209
ARCON
SFTON3D P024
SMOVL C00210 BC00210 V=11.7  +MOVJ EC00210
SMOVC C00211 BC00211 V=15.0  +MOVJ EC00211
SMOVC C00212 BC00212 V=15.0  +MOVJ EC00212
SMOVC C00213 BC00213 V=15.0  +MOVJ EC00213
SFTON3D P023
SMOVL C00214 BC00214 V=11.7  +MOVJ EC00214
SMOVL C00215 BC00215 V=11.7  +MOVJ EC00215
SMOVC C00216 BC00216 V=15.0  +MOVJ EC00216
SMOVC C00217 BC00217 V=15.0  +MOVJ EC00217
SMOVC C00218 BC00218 V=15.0  +MOVJ EC00218
ARCOF
SMOVL C00219 BC00219 V=166.7  +MOVJ EC00219
SFTOF3D
SMOVL C00220 BC00220 V=666.7  +MOVJ EC00220
SFTON3D P031
SMOVL C00221 BC00221 V=666.7  +MOVJ EC00221
SMOVL C00222 BC00222 V=166.7 PL=0  +MOVJ EC00222
SREFP 1 C00223 BC00223  +REFP EC00223
SREFP 2 C00224 BC00224  +REFP EC00224
ARCON
SWVON WEV#(71)
SMOVL C00225 BC00225 V=6.7  +MOVJ EC00225
ARCOF
SWVOF
SMOVL C00226 BC00226 V=166.7  +MOVJ EC00226
SMOVL C00227 BC00227 V=166.7  +MOVJ EC00227
SMOVL C00228 BC00228 V=166.7 PL=0  +MOVJ EC00228
ARCON
SWVON WEV#(70)
SMOVL C00229 BC00229 V=6.7  +MOVJ EC00229
SFTON3D P032
SMOVL C00230 BC00230 V=6.7  +MOVJ EC00230
ARCOF
SWVOF
SMOVL C00231 BC00231 V=33.3 PL=0  +MOVJ EC00231
ARCON
SWVON WEV#(70)
SMOVL C00232 BC00232 V=6.7  +MOVJ EC00232
ARCOF
SWVOF
SMOVL C00233 BC00233 V=166.7  +MOVJ EC00233
SFTOF3D
SMOVL C00234 BC00234 V=166.7  +MOVJ EC00234
SMOVL C00235 BC00235 V=166.7  +MOVJ EC00235
SFTON3D P027
SMOVL C00236 BC00236 V=166.7 PL=0  +MOVJ EC00236
ARCON
SMOVL C00237 BC00237 V=11.7  +MOVJ EC00237
SMOVC C00238 BC00238 V=15.0  +MOVJ EC00238
SMOVC C00239 BC00239 V=15.0  +MOVJ EC00239
SFTON3D P026
SMOVC C00240 BC00240 V=15.0  +MOVJ EC00240
SMOVL C00241 BC00241 V=11.7  +MOVJ EC00241
SFTON3D P025
SMOVL C00242 BC00242 V=11.7  +MOVJ EC00242
ARCOF
SMOVL C00243 BC00243 V=166.7  +MOVJ EC00243
SFTOF3D
SMOVL C00244 BC00244 V=666.7  +MOVJ EC00244
SMOVL C00245 BC00245 V=666.7  +MOVJ EC00245
SFTON3D P022
SMOVL C00246 BC00246 V=166.7 PL=0  +MOVJ EC00246
ARCON
SFTON3D P021
SMOVL C00247 BC00247 V=11.7  +MOVJ EC00247
SMOVC C00248 BC00248 V=15.0  +MOVJ EC00248
SMOVC C00249 BC00249 V=15.0  +MOVJ EC00249
SMOVC C00250 BC00250 V=15.0  +MOVJ EC00250
SFTON3D P022
SMOVL C00251 BC00251 V=11.7  +MOVJ EC00251
SMOVL C00252 BC00252 V=11.7  +MOVJ EC00252
SMOVC C00253 BC00253 V=15.0  +MOVJ EC00253
SMOVC C00254 BC00254 V=15.0  +MOVJ EC00254
SMOVC C00255 BC00255 V=15.0  +MOVJ EC00255
ARCOF
SMOVL C00256 BC00256 V=166.7  +MOVJ EC00256
SFTOF3D
MOVL C00257 BC00257 V=666.7  +MOVJ EC00257 VJ=0.78
MOVL C00258 BC00258 V=666.7  +MOVJ EC00258 VJ=0.78
SFTON3D P035
SMOVL C00259 BC00259 V=166.7 PL=0  +MOVJ EC00259
ARCON
SMOVL C00260 BC00260 V=11.7  +MOVJ EC00260
SMOVL C00261 BC00261 V=11.7  +MOVJ EC00261
SFTON3D P036
SMOVL C00262 BC00262 V=11.7  +MOVJ EC00262
SMOVC C00263 BC00263 V=15.0  +MOVJ EC00263
SMOVC C00264 BC00264 V=15.0  +MOVJ EC00264
SFTON3D P037
SMOVC C00265 BC00265 V=15.0  +MOVJ EC00265
SMOVL C00266 BC00266 V=11.7  +MOVJ EC00266
SMOVL C00267 BC00267 V=11.7  +MOVJ EC00267
SFTON3D P038
COMM SMOVL C00268 BC00268 V=11.7  +MOVJ EC00268
SMOVL C00269 BC00269 V=13.3  +MOVJ EC00269
ARCOF
SMOVL C00270 BC00270 V=166.7  +MOVJ EC00270
SFTOF3D
SMOVL C00271 BC00271 V=666.7  +MOVJ EC00271
SMOVL C00272 BC00272 V=666.7  +MOVJ EC00272
SMOVL C00273 BC00273 V=666.7  +MOVJ EC00273
SFTON3D P027
SMOVL C00274 BC00274 V=166.7 PL=0  +MOVJ EC00274
ARCON
SMOVL C00275 BC00275 V=11.7  +MOVJ EC00275
SFTON3D P028
SMOVL C00276 BC00276 V=11.7  +MOVJ EC00276
SMOVL C00277 BC00277 V=11.7  +MOVJ EC00277
ARCOF
SMOVL C00278 BC00278 V=166.7  +MOVJ EC00278
SFTOF3D
SMOVL C00279 BC00279 V=666.7  +MOVJ EC00279
MOVJ C00280 BC00280 VJ=100.00  +MOVJ EC00280 VJ=100.00
'
END
